SYSTEM ROBOT_HMI (* System Configuration *)
  (* Standard: 61499-1 *)
  (* Version 0.3, 2003-12-05, JHC, Rockwell Automation, Renamed from NEWSYSTEM. *)
  (* Version 0.2, 2002-11-05, JHC, Rockwell Automation, Fixed missing (empty) FBD in Application. *)
  (* Version 0.1, 2002-01-17, JHC, Rockwell Automation, Minor cleanup *)
  (* Version 0.0, 2000-05-27, JHC, Rockwell Automation *)
  APPLICATION APP1
  END_APPLICATION
  DEVICE ROBOT_HMI_DEVICE : FRAME_DEVICE(BOUNDS := [1100,300,600,400], GRID := [1,1])
    RESOURCE ROBOT_HMI_PROCESSOR : PANEL_RESOURCE(ROWS := 11, COLS := 2)
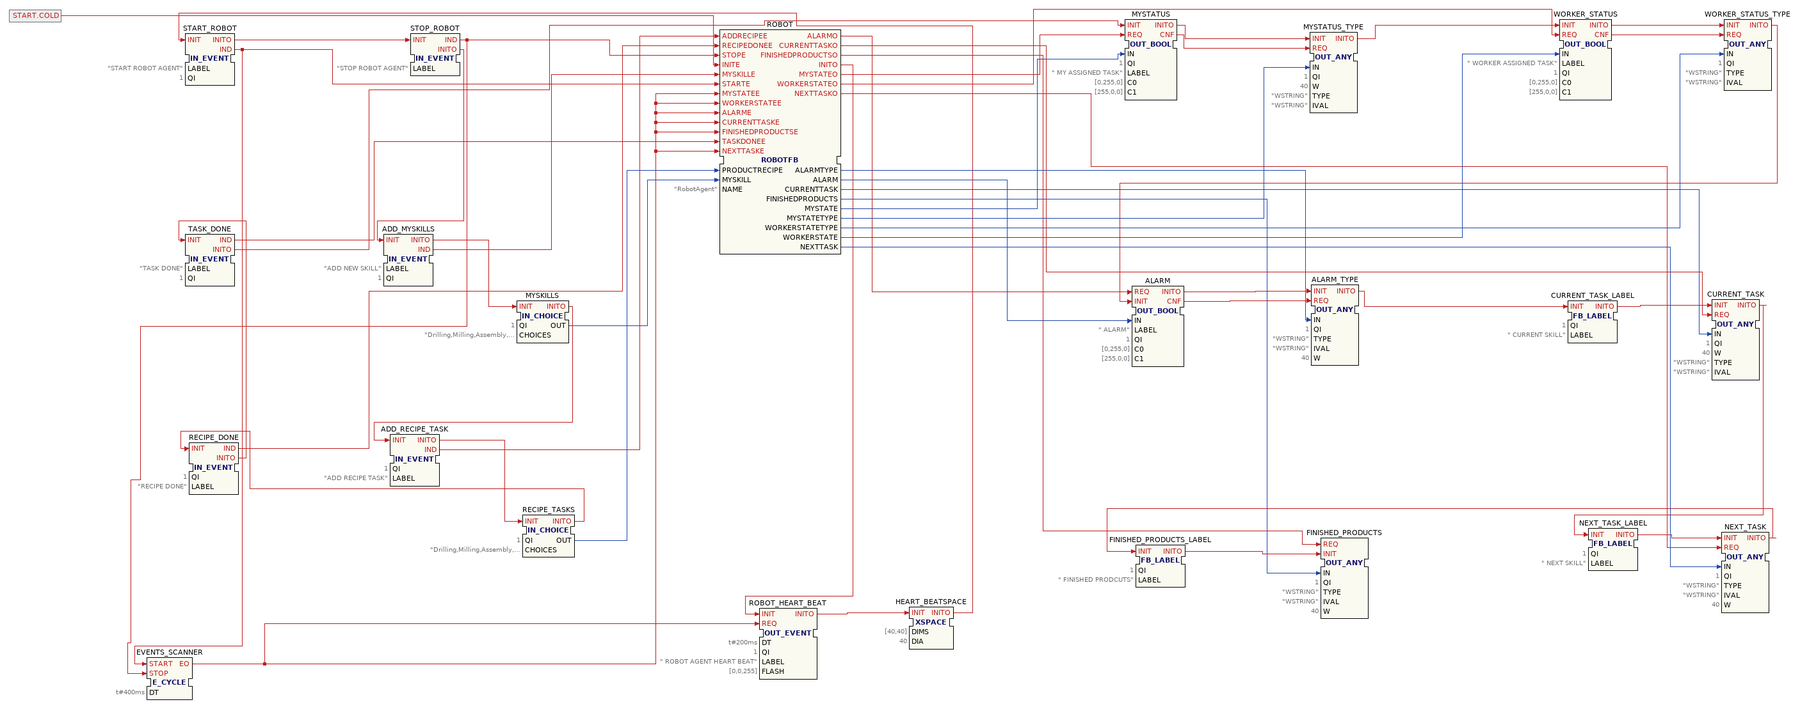
      FBS
        ROBOT : ROBOTFB(NAME := "RobotAgent");
        ADD_RECIPE_TASK : IN_EVENT(QI := 1, LABEL := "ADD RECIPE TASK");
        RECIPE_TASKS : IN_CHOICE(QI := 1, CHOICES := "Drilling,Milling,Assembly,Painting,Shaping");
        RECIPE_DONE : IN_EVENT(QI := 1, LABEL := "RECIPE DONE");
        MYSTATUS_TYPE : OUT_ANY(QI := 1, W := 40, TYPE := "WSTRING", IVAL := "WSTRING");
        ALARM_TYPE : OUT_ANY(QI := 1, TYPE := "WSTRING", IVAL := "WSTRING", W := 40);
        ALARM : OUT_BOOL(LABEL := "                      ALARM", QI := 1, C0 := [0,255,0], C1 := [255,0,0]);
        CURRENT_TASK_LABEL : FB_LABEL(QI := 1, LABEL := "                     CURRENT SKILL");
        CURRENT_TASK : OUT_ANY(QI := 1, W := 40, TYPE := "WSTRING", IVAL := "WSTRING");
        FINISHED_PRODUCTS_LABEL : FB_LABEL(QI := 1, LABEL := "                FINISHED PRODCUTS");
        FINISHED_PRODUCTS : OUT_ANY(QI := 1, TYPE := "WSTRING", IVAL := "WSTRING", W := 40);
        WORKER_STATUS_TYPE : OUT_ANY(QI := 1, TYPE := "WSTRING", IVAL := "WSTRING");
        START_ROBOT : IN_EVENT(LABEL := "START ROBOT AGENT", QI := 1);
        STOP_ROBOT : IN_EVENT(LABEL := "STOP ROBOT AGENT");
        ADD_MYSKILLS : IN_EVENT(LABEL := "ADD NEW SKILL", QI := 1);
        MYSKILLS : IN_CHOICE(QI := 1, CHOICES := "Drilling,Milling,Assembly,Painting,Shaping");
        ROBOT_HEART_BEAT : OUT_EVENT(DT := t#200ms, QI := 1, LABEL := "                 ROBOT AGENT HEART BEAT", FLASH := [0,0,255]);
        EVENTS_SCANNER : E_CYCLE(DT := t#400ms);
        HEART_BEATSPACE : XSPACE(DIMS := [40,40], DIA := 40);
        TASK_DONE : IN_EVENT(LABEL := "TASK DONE", QI := 1);
        MYSTATUS : OUT_BOOL(QI := 1, LABEL := "           MY ASSIGNED TASK", C0 := [0,255,0], C1 := [255,0,0]);
        WORKER_STATUS : OUT_BOOL(LABEL := "      WORKER ASSIGNED TASK", QI := 1, C0 := [0,255,0], C1 := [255,0,0]);
        NEXT_TASK_LABEL : FB_LABEL(QI := 1, LABEL := "                        NEXT SKILL");
        NEXT_TASK : OUT_ANY(QI := 1, TYPE := "WSTRING", IVAL := "WSTRING", W := 40);
      END_FBS
      EVENT_CONNECTIONS
        ADD_RECIPE_TASK.INITO TO RECIPE_TASKS.INIT;
        ADD_RECIPE_TASK.IND TO ROBOT.ADDRECIPEE;
        RECIPE_TASKS.INITO TO RECIPE_DONE.INIT;
        RECIPE_DONE.IND TO ROBOT.RECIPEDONEE;
        ALARM.INITO TO ALARM_TYPE.INIT;
        ROBOT.ALARMO TO ALARM.REQ;
        ALARM_TYPE.INITO TO CURRENT_TASK_LABEL.INIT;
        CURRENT_TASK_LABEL.INITO TO CURRENT_TASK.INIT;
        ALARM.CNF TO ALARM_TYPE.REQ;
        ROBOT.CURRENTTASKO TO CURRENT_TASK.REQ;
        ROBOT.FINISHEDPRODUCTSO TO FINISHED_PRODUCTS.REQ;
        FINISHED_PRODUCTS_LABEL.INITO TO FINISHED_PRODUCTS.INIT;
        WORKER_STATUS_TYPE.INITO TO ALARM.INIT;
        START_ROBOT.INITO TO STOP_ROBOT.INIT;
        STOP_ROBOT.IND TO ROBOT.STOPE;
        START.COLD TO ROBOT.INITE;
        ADD_MYSKILLS.INITO TO MYSKILLS.INIT;
        ADD_MYSKILLS.IND TO ROBOT.MYSKILLE;
        STOP_ROBOT.INITO TO ADD_MYSKILLS.INIT;
        MYSKILLS.INITO TO ADD_RECIPE_TASK.INIT;
        ROBOT_HEART_BEAT.INITO TO HEART_BEATSPACE.INIT;
        HEART_BEATSPACE.INITO TO START_ROBOT.INIT;
        ROBOT.INITO TO ROBOT_HEART_BEAT.INIT;
        START_ROBOT.IND TO ROBOT.STARTE;
        START_ROBOT.IND TO EVENTS_SCANNER.START;
        STOP_ROBOT.IND TO EVENTS_SCANNER.STOP;
        EVENTS_SCANNER.EO TO ROBOT_HEART_BEAT.REQ;
        EVENTS_SCANNER.EO TO ROBOT.MYSTATEE;
        EVENTS_SCANNER.EO TO ROBOT.WORKERSTATEE;
        EVENTS_SCANNER.EO TO ROBOT.ALARME;
        EVENTS_SCANNER.EO TO ROBOT.CURRENTTASKE;
        EVENTS_SCANNER.EO TO ROBOT.FINISHEDPRODUCTSE;
        RECIPE_DONE.INITO TO TASK_DONE.INIT;
        TASK_DONE.IND TO ROBOT.TASKDONEE;
        TASK_DONE.INITO TO MYSTATUS.INIT;
        MYSTATUS.INITO TO MYSTATUS_TYPE.INIT;
        ROBOT.MYSTATEO TO MYSTATUS.REQ;
        MYSTATUS.CNF TO MYSTATUS_TYPE.REQ;
        MYSTATUS_TYPE.INITO TO WORKER_STATUS.INIT;
        WORKER_STATUS.INITO TO WORKER_STATUS_TYPE.INIT;
        ROBOT.WORKERSTATEO TO WORKER_STATUS.REQ;
        WORKER_STATUS.CNF TO WORKER_STATUS_TYPE.REQ;
        EVENTS_SCANNER.EO TO ROBOT.NEXTTASKE;
        CURRENT_TASK.INITO TO NEXT_TASK_LABEL.INIT;
        NEXT_TASK_LABEL.INITO TO NEXT_TASK.INIT;
        ROBOT.NEXTTASKO TO NEXT_TASK.REQ;
        NEXT_TASK.INITO TO FINISHED_PRODUCTS_LABEL.INIT;
      END_CONNECTIONS
      DATA_CONNECTIONS
        RECIPE_TASKS.OUT TO ROBOT.PRODUCTRECIPE;
        ROBOT.ALARMTYPE TO ALARM_TYPE.IN;
        ROBOT.ALARM TO ALARM.IN;
        ROBOT.CURRENTTASK TO CURRENT_TASK.IN;
        ROBOT.FINISHEDPRODUCTS TO FINISHED_PRODUCTS.IN;
        MYSKILLS.OUT TO ROBOT.MYSKILL;
        ROBOT.MYSTATE TO MYSTATUS.IN;
        ROBOT.MYSTATETYPE TO MYSTATUS_TYPE.IN;
        ROBOT.WORKERSTATETYPE TO WORKER_STATUS_TYPE.IN;
        ROBOT.WORKERSTATE TO WORKER_STATUS.IN;
        ROBOT.NEXTTASK TO NEXT_TASK.IN;
      END_CONNECTIONS
    END_RESOURCE
  END_DEVICE
END_SYSTEM
